Staubli VAL3: encodeHeader.pgx

program encodeHeader(MessageHeader& x_header, num& x_nData[], bool& x_bError)
  local num l_nIndexOffset
begin
  // Copyright 2025 ICUBE Laboratory, University of Strasbourg
  //
  // Licensed under the Apache License, Version 2.0 (the "License");
  // you may not use this file except in compliance with the License.
  // You may obtain a copy of the License at
  //
  //     http://www.apache.org/licenses/LICENSE-2.0
  //
  // Unless required by applicable law or agreed to in writing, software
  // distributed under the License is distributed on an "AS IS" BASIS,
  // WITHOUT WARRANTIES OR CONDITIONS OF ANY KIND, either express or implied.
  // See the License for the specific language governing permissions and
  // limitations under the License.

  // Check header is well structured
  if(x_header.nMsgSequenceNumber < 0)
    x_bError = true
    logMsg("ros2_server::encodeHeader : Error, invalid (negative) sequence number",2)
    return
  endIf

  if(size(x_nData)==1)
    x_bError = true
    logMsg("ros2_server::encodeHeader : Error, data buffer not initialized (size is 1)",2)
    return
  endIf

  if(size(x_nData)<x_header.nHeaderSize)
    x_bError = true
    logMsg("ros2_server::encodeHeader : Error, invalid data size",2)
    return
  endIf

  // Serialization
  // uint8_t   <-> "1" Unsigned byte
  // uint16_t  <-> "2l" Unsigned word, little endian
  // float32_t <-> "4.0l" Single precision floating point value, little endian

  l_nIndexOffset = 0
  toBinary(x_header.nMagicNumber,2,"2l",x_nData[l_nIndexOffset])
  l_nIndexOffset = l_nIndexOffset + 2
  toBinary(x_header.nProtocolVersion,1,"1",x_nData[l_nIndexOffset])
  l_nIndexOffset = l_nIndexOffset + 1
  toBinary(x_header.nMsgType,1, "1",x_nData[l_nIndexOffset])
  l_nIndexOffset = l_nIndexOffset + 1
  toBinary(x_header.nMsgSequenceNumber,2,"2l",x_nData[l_nIndexOffset])
  l_nIndexOffset = l_nIndexOffset + 2
  toBinary(x_header.nMsgSequenceNumber,2,"2l",x_nData[l_nIndexOffset])
  l_nIndexOffset = l_nIndexOffset + 2

  if(l_nIndexOffset != x_header.nHeaderSize)
    x_bError = true
    logMsg("ros2_server::encodeHeader : Error, binary encoding failed",2)
    return
  endIf

  // OK
  x_bError = false
end
